(* IEC 61131-3 sources: EnigmaLogic-Roomcontroller/PID, 6 files *)

(* ---- PIC02.ST ---- *)
PROGRAM PIC02
VAR_EXTERNAL
DisplayAddress : usint;
DisplayPoint74 : real;

SI01 : real;
SI02 : real;
SI03 : real;
SI04 : real;

PI01 : real;
PI02 : real;
PI03 : real;
PI04 : real;

HE01 : BOOL;
CO01 : BOOL;

END_VAR

VAR
PID_CONTROL : PIDFB ; (* The functionblock type: PIDFB *)
in01 : real;
var01 : real := 0.0;
var02 : real := 0.0;
var03 : real := 10.0;
var04 : real := 2000.0;
cal01 : real;
cal02 : real;
cal03 : real;
cal04 : real;
cal05 : real;
Result : word;
Result2 : int;
y01 : real := 0.0;
y02 : real := 100.0;
x01 : real := 0.0;
x02 : real;
in02 : real;
min01 : real := 0.0;
max01 : real  := 2000.0;
min02 : real := 0.0;
max02 : real  := 50.0;

END_VAR
(*Setpoint calculator C02*)
in01 := WORD_TO_REAL (GetRegisterF(RegNumber:=508)); (*AI09 == CO2 0-10V)*)
 cal01 := var03 - var01;
 cal02 := var02 - var04;
 cal03 := cal02 / cal01;
 cal04 := in01 - var01;
 cal05 := var02 - (cal04 * cal03);

IF var02 = var04 THEN
   cal05 := in01;
END_IF;

 cal05 := LIMIT(min01,cal05,max01);

PID_CONTROL.measurement := cal05;
PID_CONTROL.setpoint := SI02; (*SI02 == Setpoint room co2 controller)*)
PID_CONTROL.stages := 1; (* INT, between 1 and 6 *)
PID_CONTROL.balance := 0; (* INT, between 0 and 6 *)
PID_CONTROL.deadzone := 50.0 ; (* REAL *)
PID_CONTROL.comfort := 0.1; (* REAL *)
PID_CONTROL.min1 := 0; (* INT, between 0 and 100 *)
PID_CONTROL.max1 := 100; (* INT, between 0 and 100 *)
PID_CONTROL.pband1 := 100.0; (* REAL, bigger than 0 *)
PID_CONTROL.iTime := 120; (* INT, seconds, bigger than 0 *)
PID_CONTROL.dTime := 0; (* INT, seconds *)
(* calling the execution of the functionblock *)
PID_CONTROL();

PI01 := PID_CONTROL.out1;
END_PROGRAM

(* ---- PIDDYN.ST ---- *)
PROGRAM PIDDYN
VAR_EXTERNAL
DisplayAddress : usint;
DisplayPoint74 : real;
DisplayPoint8 : real;

SI01 : real;
SI02 : real;
SI03 : real;
SI04 : real;

PI01 : real;
PI02 : real;
PI03 : real;
PI04 : real;

HE01 : BOOL;
CO01 : BOOL;

END_VAR

VAR
PID_CONTROL : PIDFB ; (* The functionblock type: PIDFB *)
in01 : real;
var01 : real := 0.0;
var02 : real := 0.0;
var03 : real := 10.0;
var04 : real := 2000.0;
cal01 : real;
cal02 : real;
cal03 : real;
cal04 : real;
cal05 : real;
Result : word;
Result2 : int;
y01 : real := 0.0;
y02 : real := 100.0;
x01 : real := 0.0;
x02 : real;
in02 : real;
min01 : real := 0.0;
max01 : real  := 2000.0;
min02 : real := 0.0;
max02 : real  := 50.0;
Output_1 : REAL ;
Output_2 : REAL ;

END_VAR

(* Heater *)

IF HE01 THEN
Output_1 := PI02;
Result2 := SetAnalogOutputF(Number:=1, Value := Output_1);

ELSE
Output_1 := 0.0; (* returns a REAL *) (*AO01 Heating*)
Result2 := SetAnalogOutputF(Number:=1, Value := Output_1);

END_IF;

IF Output_1 > 1.0 THEN
Result2 := SetDigitalOutputF(Number:=1, Value := 10);
Result2 := SetDigitalOutputF(Number:=2, Value := 10);
ELSE
Result2 := SetDigitalOutputF(Number:=1, Value := 0);
Result2 := SetDigitalOutputF(Number:=2, Value := 0);
END_IF;

(* Cooler  *)

IF CO01 THEN
Output_2 := PI03; (* returns a REAL *) (*AO02 Cooling*)
Result2 := SetAnalogOutputF(Number:=2, Value := Output_2);

ELSE
Output_2 := 0.0; (* returns a REAL *) (*AO02 Cooling*)
Result2 := SetAnalogOutputF(Number:=2, Value := Output_2);

END_IF;

(* Heating - Cooling on Display *)

DisplayPoint8 := GetDisplayPointValueF(PointNumber:=8, SlaveAddress:=DisplayAddress, OldValue:=DisplayPoint8);
IF Output_1 > 10.0 THEN
	DisplayPoint8 := 1.0;

ELSIF Output_2 > 10.0 THEN
	DisplayPoint8 := 2.0;

ELSE
	DisplayPoint8 := 0.0;

END_IF;

Result2 := SetDisplayPointF(PointNumber:=8, PointType:=0, PointUnit:=0, SlaveAddress:=DisplayAddress, PointValue:=DisplayPoint8 );

(*in02 := MAX(Output_1,PI01,Output_2);*)
in02 := MAX(Output_1,Output_2);

(* POINT74: max *)
DisplayPoint74 := GetDisplayPointValueF(PointNumber:=74, SlaveAddress:=DisplayAddress, OldValue:=DisplayPoint74);
Result2 := SetDisplayPointF(PointNumber:=74, PointType:=0, PointUnit:=0, SlaveAddress:=DisplayAddress, PointValue:=DisplayPoint74 );

x02 := DisplayPoint74;

(*Setpoint calculator MAX VAV*)
 cal01 := y02 - y01;
 cal02 := x01 - x02;
 cal03 := cal02 / cal01;
 cal04 := in02 - y01;
 PI04 := x01 - (cal04 * cal03);

PI04 := LIMIT(min02,PI04,x02);
Result2 := SetAnalogOutputF(Number:=3, Value := PI04);
END_PROGRAM

(* ---- PIDEA.ST ---- *)
PROGRAM PIDEA
VAR_EXTERNAL
SI01 : real;
SI02 : real;
SI03 : real;
SI04 : real;

PI01 : real;
PI02 : real;

END_VAR

VAR
PID_CONTROL : PIDFB ; (* The functionblock type: PIDFB *)
Output_4 : REAL ;
Result : int;
END_VAR

PID_CONTROL.measurement := WORD_TO_REAL(GetRegisterF(RegNumber:=507))*10.0; (*AI08 == EA Volume 0-10V)*)
PID_CONTROL.setpoint := PI02; (*PIDGLOBAL)*)
PID_CONTROL.stages := 1; (* INT, between 1 and 6 *)
PID_CONTROL.balance := 0; (* INT, between 0 and 6 *)
PID_CONTROL.deadzone := 50.0 ; (* REAL *)
PID_CONTROL.comfort := 0.1; (* REAL *)
PID_CONTROL.min1 := 0; (* INT, between 0 and 100 *)
PID_CONTROL.max1 := 100; (* INT, between 0 and 100 *)
PID_CONTROL.pband1 := 100.0; (* REAL, bigger than 0 *)
PID_CONTROL.iTime := 60; (* INT, seconds, bigger than 0 *)
PID_CONTROL.dTime := 0; (* INT, seconds *)
(* calling the execution of the functionblock *)
PID_CONTROL();
(* now we can use the output values *)

Output_4 := PID_CONTROL.out1 ; (* returns a REAL *)
Result := SetAnalogOutputF(Number:=4, Value := Output_4);
END_PROGRAM

(* ---- PIDHC.ST ---- *)
PROGRAM PIDHC
VAR_EXTERNAL
SI01 : real;
SI02 : real;
SI03 : real;
SI04 : real;

HE01 : BOOL;
CO01 : BOOL;

PI01 : real;
PI02 : real;
PI03 : real;
PI04 : real;

DisplayAddress : usint;
DisplayPoint1 : real;
DisplayPoint8 : real;
DisplayPoint10 : real;

END_VAR

VAR
PID_CONTROL : PIDFB ; (* The functionblock type: PIDFB *)
Output_1 : REAL ;
Output_2 : REAL ;
Result : int;
Result2 : real;
Result3 : real;
SetpointRT : real;
Roomtemp : real;
END_VAR

(*-------------------------------------------------------------------------------------------------------------------------------------*)
(* SET RT + ADJUST *)
Result2 := SI01;
Result3 := GetDisplayPointValueF(PointNumber:=2, SlaveAddress:=DisplayAddress, OldValue:=Result3);

IF GetRegisterF(RegNumber:=524) <> 0 THEN
	Result3 :=0.0;
	Result := SetDisplayPointF(PointNumber:=2, PointType:=0, PointUnit:=0, SlaveAddress:=DisplayAddress, PointValue:=Result3 );
	Result := SetRegisterF(RegNumber := 524, RegValue := 0);
END_IF;

(* POINT1: SET RT -> PIDHC *)
SetpointRT := GetDisplayPointValueF(PointNumber:=1, SlaveAddress:=DisplayAddress, OldValue:=SetpointRT);
SetpointRT := Result2 + Result3;
Result := SetDisplayPointF(PointNumber:=1, PointType:=1, PointUnit:=1, SlaveAddress:=DisplayAddress, PointValue:=SetpointRT );

(*-------------------------------------------------------------------------------------------------------------------------------------*)
(* POINT10: RT + Damping*)
DisplayPoint10 := GetDisplayPointValueF(PointNumber:=10, SlaveAddress:=DisplayAddress, OldValue:=DisplayPoint10);
Roomtemp := WORD_TO_REAL(GetRegisterF(RegNumber:=1013))/10.0;

IF (SetpointRT  - 0.3) < Roomtemp AND (SetpointRT  + 0.3) > Roomtemp THEN
	Roomtemp := SetpointRT;
END_IF;

Result := SetDisplayPointF(PointNumber:=10, PointType:=1, PointUnit:=0, SlaveAddress:=DisplayAddress, PointValue:=Roomtemp);
(*-------------------------------------------------------------------------------------------------------------------------------------*)

PID_CONTROL.measurement := WORD_TO_REAL(GetRegisterF(RegNumber:=1013))/10.0;
PID_CONTROL.setpoint := SetpointRT ;
PID_CONTROL.stages := 2; (* INT, between 1 and 6 *)
PID_CONTROL.balance := 1; (* INT, between 0 and 6 *)
PID_CONTROL.deadzone := 0.5 ; (* REAL *)
PID_CONTROL.comfort := 0.1; (* REAL *)
PID_CONTROL.min1 := 0; (* INT, between 0 and 100 *)
PID_CONTROL.max1 := 100; (* INT, between 0 and 100 *)
PID_CONTROL.min2 := 0; (* INT, between 0 and 100 *)
PID_CONTROL.max2 := 100; (* INT, between 0 and 100 *)
PID_CONTROL.pband1 := 20.0; (* REAL, bigger than 0 *)
PID_CONTROL.pband2 := 20.0; (* REAL, bigger than 0 *)
PID_CONTROL.iTime := 120; (* INT, seconds, bigger than 0 *)
PID_CONTROL.dTime := 0; (* INT, seconds *)
(* calling the execution of the functionblock *)
PID_CONTROL();

(* Heater *)
PI02 := PID_CONTROL.out2 ; (* returns a REAL *) (*AO01 Heating*)

(* Cooler  *)
PI03 := PID_CONTROL.out1 ; (* returns a REAL *) (*AO02 Cooling*)
END_PROGRAM

(* ---- PIDSA.ST ---- *)
PROGRAM PIDSA
VAR_EXTERNAL
SI01 : real;
SI02 : real;
SI03 : real;
SI04 : real;

PI04 : real;
END_VAR

VAR
Output_3 : REAL ;
Result : int;
END_VAR
;
END_PROGRAM

(* ---- PIDSET.ST ---- *)
PROGRAM PIDSET
VAR_EXTERNAL
SI01 : real;
SI02 : real;
SI03 : real;
SI04 : real;

HE01 : BOOL;
CO01 : BOOL;
END_VAR

VAR
result : int;

END_VAR
SI01 := WORD_TO_REAL(GetRegisterF(RegNumber:=512)); (*SI01 == Setpoint room temperature controller)*)
Result := SetRegisterF(RegNumber := 512, RegValue := REAL_TO_WORD(SI01));

SI02 := WORD_TO_REAL(GetRegisterF(RegNumber:=513)); (*SI02 == Setpoint room c02 controller)*)
Result := SetRegisterF(RegNumber := 513, RegValue := REAL_TO_WORD(SI02));

SI03 := WORD_TO_REAL(GetRegisterF(RegNumber:=514)); (*SI03 == )*)
Result := SetRegisterF(RegNumber := 514, RegValue := REAL_TO_WORD(SI03));

SI04 := WORD_TO_REAL(GetRegisterF(RegNumber:=515)); (*SI04 == )*)
Result := SetRegisterF(RegNumber := 515, RegValue := REAL_TO_WORD(SI04));

HE01 := WORD_TO_BOOL(GetRegisterF(RegNumber:=516)); (*HE01 == Heat available*)
Result := SetRegisterF(RegNumber := 516, RegValue := BOOL_TO_WORD(HE01));

CO01 := WORD_TO_BOOL(GetRegisterF(RegNumber:=517)); (*CO01 == Cool available*)
Result := SetRegisterF(RegNumber := 517, RegValue := BOOL_TO_WORD(CO01));
END_PROGRAM
